FUNCTION_BLOCK SUB_INT (* IEC 61131-3 INT Subtraction *)
  (* Standard: 61131-3 *)
  (* Version 0.0, 2004-12-15, JHC, Rockwell Automation, Converted from SRC format. *)
  (* Compiler header: package fb.rt.plc.math; *)
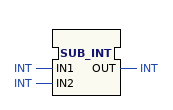
  VAR_INPUT
    IN1 : INT; (* Minuend *)
    IN2 : INT; (* Subtrahend *)
  END_VAR
  VAR_OUTPUT
    OUT : INT; (* Difference *)
  END_VAR
END_FUNCTION_BLOCK
